TYPE SCARAFITTI :
STRUCT
	parada : BOOL;
	simulacion_alfa : BOOL;
	simulacion_beta : BOOL;
	quieto : BOOL;
	en_objetivo : BOOL;
	error_objetivo : BOOL;
	ADSCOM_ready : BOOL;
END_STRUCT
END_TYPE

(* stored: Version 1.1.0.1, ProductVersion 3.1.4024.4
   DUT SCARAFITTI: Id {0d690a72-be0d-46c8-89d9-27373503178a} *)
